TYPE JBOX_Port_Map :
STRUCT
	JBOX_PORT : STRING(5);
	TESTER_PORT : STRING(5);
END_STRUCT
END_TYPE

(* stored: Version 1.1.0.1, ProductVersion 3.1.4024.10
   DUT JBOX_Port_Map: Id {cce2fca4-8635-4e79-a8ec-4f7d44b41631} *)
